TYPE strSenddata  :
	STRUCT
		STACK		: ARRAY  [0 .. 31] OF BOOL;
	END_STRUCT
END_TYPE

(* stored: Version 1.1.0.1, ProductVersion 3.1.4024.12
   DUT strSenddata: Id {ce8fb777-c09a-4c69-bfb3-d28524e3c1a7} *)
